TYPE ST_TopMoldErrors :
STRUCT
	Hydraulic					: ST_HydraulicErrorsAnalog;
	HeatingZone 				: ARRAY [1..6] OF ST_HeatingZoneErrors;
END_STRUCT
END_TYPE

(* stored: Version 1.1.0.1, ProductVersion 3.1.4020.12
   DUT ST_TopMoldErrors: Id {eb254765-a280-4d1d-9007-86666deae5e0} *)
